INTERFACE I_Signal EXTENDS Debug.I_Debug, Tags.I_Tagged

METHOD Pair : Results.Result
VAR_INPUT
	iReceiver		: I_Receiver;
END_VAR
END_METHOD

METHOD Unpair : Results.Result
VAR_INPUT
	iReceiver		: I_Receiver;
END_VAR
END_METHOD

END_INTERFACE

(* stored: Version 1.1.0.1
   Itf I_Signal: Id {da99b9e3-0afd-4c76-be10-3f8e5330abc4}
   Method Pair: Id {2bd6fd88-408d-401d-bd81-6a8cadb6efb1}
   Method Unpair: Id {0461601a-cc8c-438c-8da1-35cc47a27c85} *)
